FUNCTION_BLOCK FB_LogPersistentStorage IMPLEMENTS I_PersistentEventStorage
VAR_INPUT
	sPathName			:STRING;
END_VAR
VAR_OUTPUT
	Error				:BOOL;
END_VAR
VAR
	fbFileOpen			:FB_FileOpen;
	fbFilePuts			:FB_FilePuts;
	fbFileClose			:FB_FileClose;
	eLogWriteState		:eWriteState;
	stEventWriteToFile	:ST_Event;
	csvString			:T_MaxString;
END_VAR

CASE eLogWriteState OF 
	eWriteState.FileOpen_TRIGGER://open file
		fbFileOpen(sNetId:='',nMode:=FOPEN_MODEAPPEND OR FOPEN_MODETEXT,
					sPathName:=sPathName,ePath:=PATH_GENERIC,bExecute:=TRUE);
		IF NOT fbFileOpen.bBusy THEN 
			IF fbFileOpen.bError THEN
				eLogWriteState:=eWriteState.ERROR;
			ELSE
				fbFileOpen(sNetId:='',bExecute:=FALSE);
				eLogWriteState:=eWriteState.WAIT_FOR_EVENT;
			END_IF
		END_IF 			
				
  
	eWriteState.WAIT_FOR_EVENT:
		//do nothing here waits for the event to trigger the new event see the store event 
		
	eWriteState.WRITE_EVENT_TRIGGER:
		csvString:=CreateLogString(stEvent:=stEventWriteToFile);
		fbFilePuts(sNetId:='',bExecute:=TRUE,sLine:=csvString,hFile:=fbFileOpen.hFile);
		IF NOT fbFilePuts.bBusy THEN 
			IF fbFilePuts.bError THEN
				eLogWriteState:=eWriteState.ERROR;
			ELSE
				fbFilePuts(sNetId:='',bExecute:=FALSE);
				eLogWriteState:=eWriteState.FILE_CLOSE_TRIGGER;
			END_IF
		END_IF
		
	eWriteState.FILE_CLOSE_TRIGGER:
		fbFileClose(bExecute:=TRUE,hFile:=fbFileOpen.hFile);
		IF NOT fbFileClose.bBusy THEN 
			IF fbFileClose.bError THEN
				eLogWriteState:=eWriteState.ERROR;
			ELSE
				fbFileClose(sNetId:='',bExecute:=FALSE);
				eLogWriteState:=eWriteState.FileOpen_TRIGGER;
			END_IF
		END_IF
		
	eWriteState.ERROR:
		Error:=TRUE;

END_CASE

METHOD PRIVATE CreateLogString : T_MaxString
VAR_INPUT
	stEvent:REFERENCE TO ST_Event;
END_VAR
VAR 
	tempString:T_MaxString;
END_VAR
tempString:=stEvent.timesatamp;
tempString:=CONCAT(CONCAT(tempString,' : '),(stEvent.EventType));
tempString:=CONCAT(CONCAT(tempString,' : '),stEvent.sEventText);
tempString:=CONCAT(tempString,'$N');
CreateLogString:=tempString;
END_METHOD

METHOD StoreEvent
VAR_INPUT
	stEvent	: ST_Event;
END_VAR
IF eLogWriteState=eWriteState.WAIT_FOR_EVENT THEN 
	eLogWriteState:=eWriteState.WRITE_EVENT_TRIGGER;
	stEventWriteToFile:=stEvent;
END_IF
END_METHOD

END_FUNCTION_BLOCK

(* stored: Version 1.1.0.1, ProductVersion 3.1.4024.6
   POU FB_LogPersistentStorage: Id {4d705625-ca1c-4754-981a-010d3fed36ea}, SpecialFunc None
   Method CreateLogString: Id {dd7c7b2a-7abf-472f-a53a-fceb044fe945}
   Method StoreEvent: Id {f27094d8-b9da-456c-a85d-cdd02f165a31} *)
